// TIA Portal V20 export
// export: Created 2025-12-01T14:56:54.1618983Z, ExportSetting None, DisplayName Totally Integrated Automation Portal, DisplayVersion V20 Update 3, DisplayName TIA Portal Openness, DisplayVersion V20 Update 3, DisplayName TIA Portal Version Control Interface, DisplayVersion V20 Update 3, DisplayName STEP 7 Professional, DisplayVersion V20 Update 3, DisplayName STEP 7 Safety, DisplayVersion V20 Update 2, DisplayName WinCC Basic/Comfort/Advanced, DisplayVersion V20 Update 3, DisplayName WinCC Professional, DisplayVersion V20 Update 3, DisplayName WinCC Unified, DisplayVersion V20 Update 3
FUNCTION_BLOCK "FB341_DesapiladorBandejas_RIANTICS"   // FB341, LAD
{ S7_Optimized_Access := 'FALSE' }
// stored: AutoNumber false, SetENOAutomatically false
   VAR_INPUT
      Maquina : UInt;   // Numero de Maquina (Mesa)
      Error_Tx : Bool;   // Error en el Tx
      EnTension : Bool;   // Existe Tension en la Maquina
      MAQx_Desabilitada : Bool;   // Config MAQ. >>> DesHabilitada
      Termico_Elevacion : Bool;   // Termico de la Elevacion
      PhsMx : Bool;
      Pos_DW : Bool;   // Posición Baja del Apilador
      Pos_MID_DW : Bool;
      Pos_MID_UP : Bool;
      Pos_UP : Bool;   // Posición Alta del Apilador
      EnMovimiento_Elevacion : Bool;   // En Movineto la Elevacion
      CargaSueltaDerecha : Bool;   // Carga Suelta en el Apilador
      CargaSueltaIzquierda : Bool;
      CargaCogidaDerecha : Bool;   // Carga Cogida en el Apilador
      CargaCogidaIzquierda : Bool;
      EnMovimiento_Horquillado : Bool;   // En Movimiento el Hoquillado
      MAQ_DejarBandejas : Bool;   // Interlock >> Dejar Bandejas
      MAQ_CogerBandejas : Bool;   // Interlock >> Coger Bandejas
      MAQ_BuscarCero : Bool;   // Interlock >> Buscar Cero
      CogiendoDerecha : Bool;
      CogiendoIzquierda : Bool;
      DejandoDerecha : Bool;
      DejandoIzquierda : Bool;
      V_TOut_Elevacion : Int := 2000;   // TimeOut del Mov. de Elevacion
      V_TOut_Horquillado : Int := 2000;   // TimeOut del Mov. de Horquillado
   END_VAR
   VAR_OUTPUT
      MAQ_DejadasBandejas : Bool;   // Interlock >> Bandejas Dejadas
      MAQ_CojidasBandejas : Bool;   // Interlock >> Bandejas Cogidas
      MAQ_CeroEncontrado : Bool;   // Interlock >> Bandejas
   END_VAR
   VAR
      AP_ET00 : Bool;
      AP_ET01 : Bool;
      AP_ET100 : Bool;
      AP_ET101 : Bool;
      AP_ET102 : Bool;
      AP_ET103 : Bool;
      AP_ET104 : Bool;
      AP_ET50 : Bool;
      AP_ET51 : Bool;
      AP_ET52 : Bool;
      AP_ET53 : Bool;
      AP_ET60 : Bool;
      AP_ET61 : Bool;
      AP_ET62 : Bool;
      AP_ET63 : Bool;
      AP_ET64 : Bool;
      AP_ET65 : Bool;
      AP_ET66 : Bool;
      MA_Motor_Elev : Bool;
      MA_Slow_Velocity : Bool;
      MA_CogerCarga : Bool;   // Cerrar Cilindros para coger la pila
      MA_DejarCarga : Bool;   // Abrir Cilindros para dejas la pila
      TMP_ReposoCargaSuelta { S7_SetPoint := 'True'} : TON_TIME;
      TMP_EnTension { S7_SetPoint := 'True'} : "FB910_CNT_UHS";
      TOut_Elevacion { S7_SetPoint := 'True'} : "FB910_CNT_UHS";
      TOut_Horquillado { S7_SetPoint := 'True'} : "FB910_CNT_UHS";
      Manual : "MoviManualMaquina_Desapilador_bandejas";
   END_VAR
   VAR_TEMP
      EstadoZona : "EstadoZona";   // Estado de Zona de la Mesa
      EstadoMAQ : "EstadoMaquina_Desapilador_bandejas";   // Estado del Vehiculo Inteliguente de la Maquina
      Aux_ET00 : Bool;
   END_VAR
BEGIN

REGION Network 1: INICIALIZAR - Recoger las Variables de Estado de la Maquina
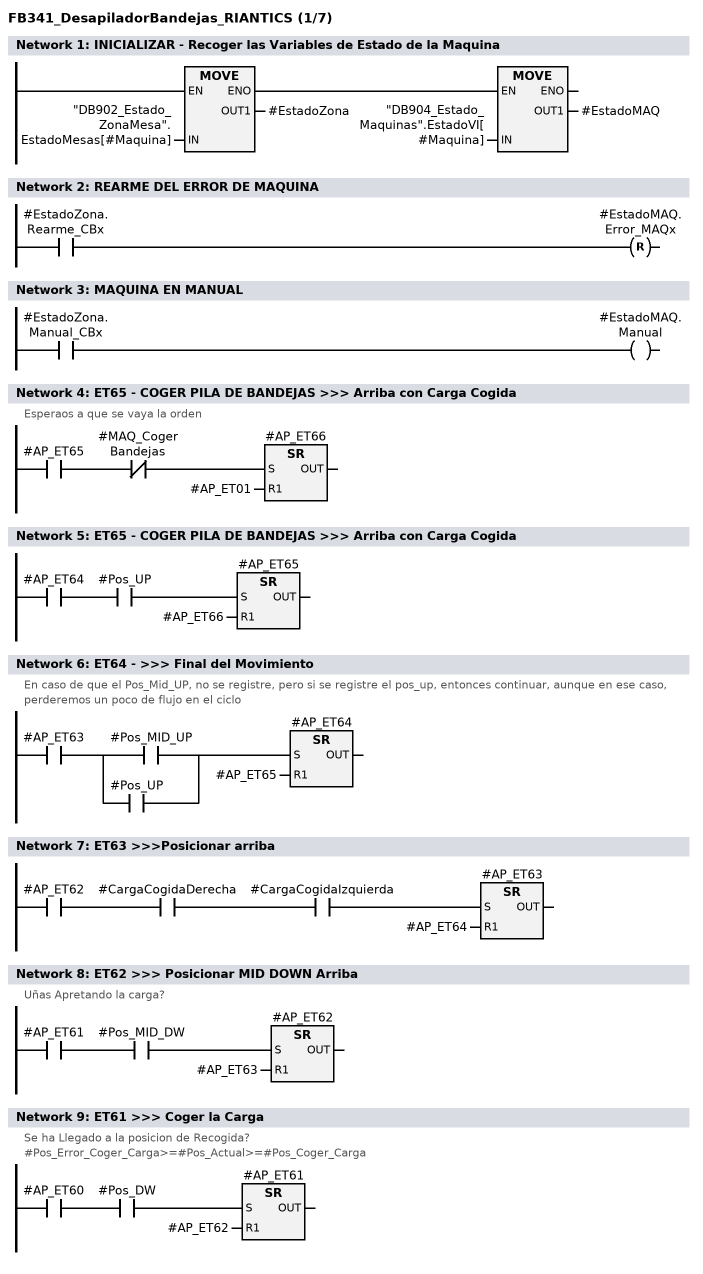
   RUNG wire#powerrail
      Move(in := "DB902_Estado_ZonaMesa".EstadoMesas[#Maquina], out1 => #EstadoZona)
      Move(in := "DB904_Estado_Maquinas".EstadoVI[#Maquina], out1 => #EstadoMAQ)
   END_RUNG
   // the same network as SCL:
   #EstadoZona := "DB902_Estado_ZonaMesa".EstadoMesas[#Maquina];
   #EstadoMAQ := "DB904_Estado_Maquinas".EstadoVI[#Maquina];
END_REGION

REGION Network 2: REARME DEL ERROR DE MAQUINA
   RUNG wire#powerrail
      Contact( #EstadoZona.Rearme_CBx )
      R_Coil( #EstadoMAQ.Error_MAQx )
   END_RUNG
   // the same network as SCL:
   IF #EstadoZona.Rearme_CBx THEN #EstadoMAQ.Error_MAQx := FALSE; END_IF;
END_REGION

REGION Network 3: MAQUINA EN MANUAL
   RUNG wire#powerrail
      Contact( #EstadoZona.Manual_CBx )
      Coil( #EstadoMAQ.Manual )
   END_RUNG
   // the same network as SCL:
   #EstadoMAQ.Manual := #EstadoZona.Manual_CBx;
END_REGION

REGION Network 4: ET65 - COGER PILA DE BANDEJAS >>> Arriba con Carga Cogida
   // Esperaos a que se vaya la orden
   RUNG wire#powerrail
      Contact( #AP_ET65 )
      I_Contact( #MAQ_CogerBandejas )
      S_SR(operand := #AP_ET66, r1 := #AP_ET01)
   END_RUNG
   // the same network as SCL:
   IF #AP_ET65 AND NOT #MAQ_CogerBandejas THEN
       #AP_ET66 := TRUE;   // SR flip-flop
   END_IF;
   IF #AP_ET01 THEN #AP_ET66 := FALSE; END_IF;
END_REGION

REGION Network 5: ET65 - COGER PILA DE BANDEJAS >>> Arriba con Carga Cogida
   RUNG wire#powerrail
      Contact( #AP_ET64 )
      Contact( #Pos_UP )
      S_SR(operand := #AP_ET65, r1 := #AP_ET66)
   END_RUNG
   // the same network as SCL:
   IF #AP_ET64 AND #Pos_UP THEN
       #AP_ET65 := TRUE;   // SR flip-flop
   END_IF;
   IF #AP_ET66 THEN #AP_ET65 := FALSE; END_IF;
END_REGION

REGION Network 6: ET64 - >>> Final del Movimiento
   // En caso de que el Pos_Mid_UP, no se registre, pero si se registre el pos_up, entonces continuar, aunque en ese caso, perderemos un poco de flujo en el ciclo
   RUNG wire#powerrail
      Contact( #AP_ET63 )
      wire#w1
      Contact( #Pos_MID_UP )
      wire#w2
      S_SR(operand := #AP_ET64, r1 := #AP_ET65)
   END_RUNG
   RUNG wire#w1
      Contact( #Pos_UP )
   END_RUNG wire#w2
   // the same network as SCL:
   IF #AP_ET63 AND (#Pos_MID_UP OR #Pos_UP) THEN
       #AP_ET64 := TRUE;   // SR flip-flop
   END_IF;
   IF #AP_ET65 THEN #AP_ET64 := FALSE; END_IF;
END_REGION

REGION Network 7: ET63 >>>Posicionar arriba
   RUNG wire#powerrail
      Contact( #AP_ET62 )
      Contact( #CargaCogidaDerecha )
      Contact( #CargaCogidaIzquierda )
      S_SR(operand := #AP_ET63, r1 := #AP_ET64)
   END_RUNG
   // the same network as SCL:
   IF #AP_ET62 AND #CargaCogidaDerecha AND #CargaCogidaIzquierda THEN
       #AP_ET63 := TRUE;   // SR flip-flop
   END_IF;
   IF #AP_ET64 THEN #AP_ET63 := FALSE; END_IF;
END_REGION

REGION Network 8: ET62 >>> Posicionar MID DOWN Arriba
   // Uñas Apretando la carga?
   RUNG wire#powerrail
      Contact( #AP_ET61 )
      Contact( #Pos_MID_DW )
      S_SR(operand := #AP_ET62, r1 := #AP_ET63)
   END_RUNG
   // the same network as SCL:
   IF #AP_ET61 AND #Pos_MID_DW THEN
       #AP_ET62 := TRUE;   // SR flip-flop
   END_IF;
   IF #AP_ET63 THEN #AP_ET62 := FALSE; END_IF;
END_REGION

REGION Network 9: ET61 >>> Coger la Carga
   // Se ha Llegado a la posicion de Recogida?
   // #Pos_Error_Coger_Carga>=#Pos_Actual>=#Pos_Coger_Carga
   RUNG wire#powerrail
      Contact( #AP_ET60 )
      Contact( #Pos_DW )
      S_SR(operand := #AP_ET61, r1 := #AP_ET62)
   END_RUNG
   // the same network as SCL:
   IF #AP_ET60 AND #Pos_DW THEN
       #AP_ET61 := TRUE;   // SR flip-flop
   END_IF;
   IF #AP_ET62 THEN #AP_ET61 := FALSE; END_IF;
END_REGION

REGION Network 10: ET60 >>> Posicionar Abajo(Anulado)
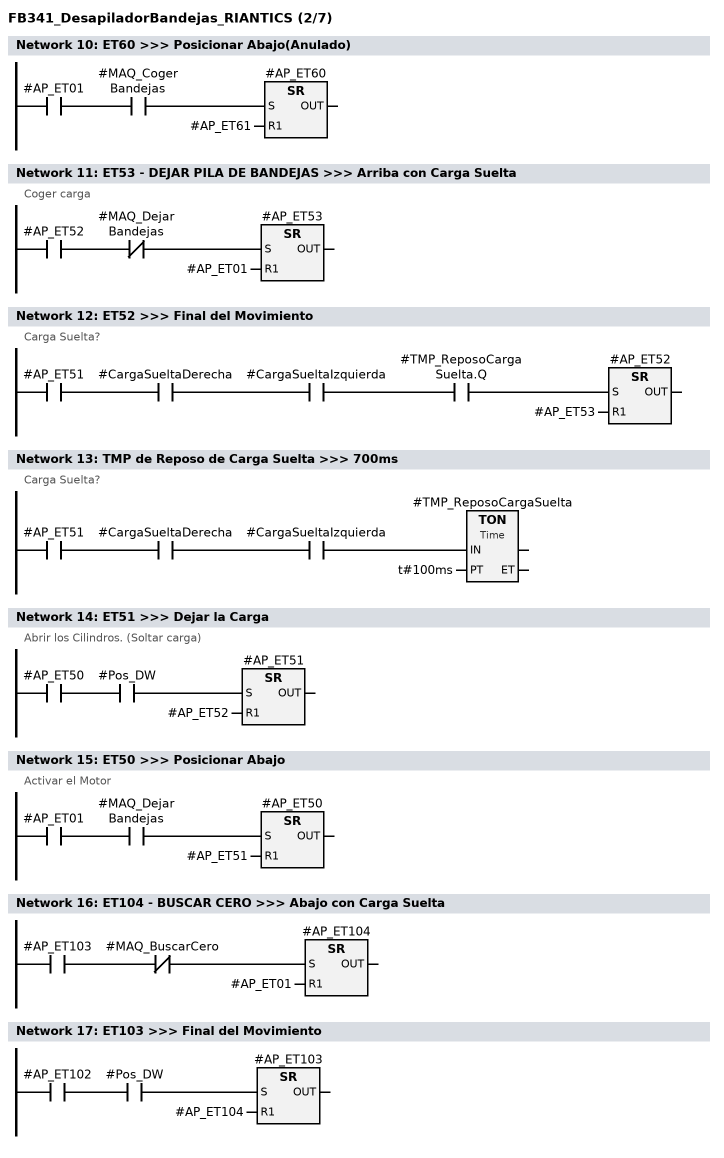
   RUNG wire#powerrail
      Contact( #AP_ET01 )
      Contact( #MAQ_CogerBandejas )
      S_SR(operand := #AP_ET60, r1 := #AP_ET61)
   END_RUNG
   // the same network as SCL:
   IF #AP_ET01 AND #MAQ_CogerBandejas THEN
       #AP_ET60 := TRUE;   // SR flip-flop
   END_IF;
   IF #AP_ET61 THEN #AP_ET60 := FALSE; END_IF;
END_REGION

REGION Network 11: ET53 - DEJAR PILA DE BANDEJAS >>> Arriba con Carga Suelta
   // Coger carga
   RUNG wire#powerrail
      Contact( #AP_ET52 )
      I_Contact( #MAQ_DejarBandejas )
      S_SR(operand := #AP_ET53, r1 := #AP_ET01)
   END_RUNG
   // the same network as SCL:
   IF #AP_ET52 AND NOT #MAQ_DejarBandejas THEN
       #AP_ET53 := TRUE;   // SR flip-flop
   END_IF;
   IF #AP_ET01 THEN #AP_ET53 := FALSE; END_IF;
END_REGION

REGION Network 12: ET52 >>> Final del Movimiento
   // Carga Suelta?
   RUNG wire#powerrail
      Contact( #AP_ET51 )
      Contact( #CargaSueltaDerecha )
      Contact( #CargaSueltaIzquierda )
      Contact( #TMP_ReposoCargaSuelta.Q )
      S_SR(operand := #AP_ET52, r1 := #AP_ET53)
   END_RUNG
   // the same network as SCL:
   IF #AP_ET51 AND #CargaSueltaDerecha AND #CargaSueltaIzquierda AND #TMP_ReposoCargaSuelta.Q THEN
       #AP_ET52 := TRUE;   // SR flip-flop
   END_IF;
   IF #AP_ET53 THEN #AP_ET52 := FALSE; END_IF;
END_REGION

REGION Network 13: TMP de Reposo de Carga Suelta >>> 700ms
   // Carga Suelta?
   RUNG wire#powerrail
      Contact( #AP_ET51 )
      Contact( #CargaSueltaDerecha )
      Contact( #CargaSueltaIzquierda )
      { S7_Templates := "time_type := Time" } #TMP_ReposoCargaSuelta.TON(pt := t#100ms, et =>)
   END_RUNG
   // the same network as SCL:
   #TMP_ReposoCargaSuelta(IN := #AP_ET51 AND #CargaSueltaDerecha AND #CargaSueltaIzquierda, PT := t#100ms);   // TON
END_REGION

REGION Network 14: ET51 >>> Dejar la Carga
   // Abrir los Cilindros. (Soltar carga)
   RUNG wire#powerrail
      Contact( #AP_ET50 )
      Contact( #Pos_DW )
      S_SR(operand := #AP_ET51, r1 := #AP_ET52)
   END_RUNG
   // the same network as SCL:
   IF #AP_ET50 AND #Pos_DW THEN
       #AP_ET51 := TRUE;   // SR flip-flop
   END_IF;
   IF #AP_ET52 THEN #AP_ET51 := FALSE; END_IF;
END_REGION

REGION Network 15: ET50 >>> Posicionar Abajo
   // Activar el Motor
   RUNG wire#powerrail
      Contact( #AP_ET01 )
      Contact( #MAQ_DejarBandejas )
      S_SR(operand := #AP_ET50, r1 := #AP_ET51)
   END_RUNG
   // the same network as SCL:
   IF #AP_ET01 AND #MAQ_DejarBandejas THEN
       #AP_ET50 := TRUE;   // SR flip-flop
   END_IF;
   IF #AP_ET51 THEN #AP_ET50 := FALSE; END_IF;
END_REGION

REGION Network 16: ET104 - BUSCAR CERO >>> Abajo con Carga Suelta
   RUNG wire#powerrail
      Contact( #AP_ET103 )
      I_Contact( #MAQ_BuscarCero )
      S_SR(operand := #AP_ET104, r1 := #AP_ET01)
   END_RUNG
   // the same network as SCL:
   IF #AP_ET103 AND NOT #MAQ_BuscarCero THEN
       #AP_ET104 := TRUE;   // SR flip-flop
   END_IF;
   IF #AP_ET01 THEN #AP_ET104 := FALSE; END_IF;
END_REGION

REGION Network 17: ET103 >>> Final del Movimiento
   RUNG wire#powerrail
      Contact( #AP_ET102 )
      Contact( #Pos_DW )
      S_SR(operand := #AP_ET103, r1 := #AP_ET104)
   END_RUNG
   // the same network as SCL:
   IF #AP_ET102 AND #Pos_DW THEN
       #AP_ET103 := TRUE;   // SR flip-flop
   END_IF;
   IF #AP_ET104 THEN #AP_ET103 := FALSE; END_IF;
END_REGION

REGION Network 18: ET102 >>> Posicionar Abajo
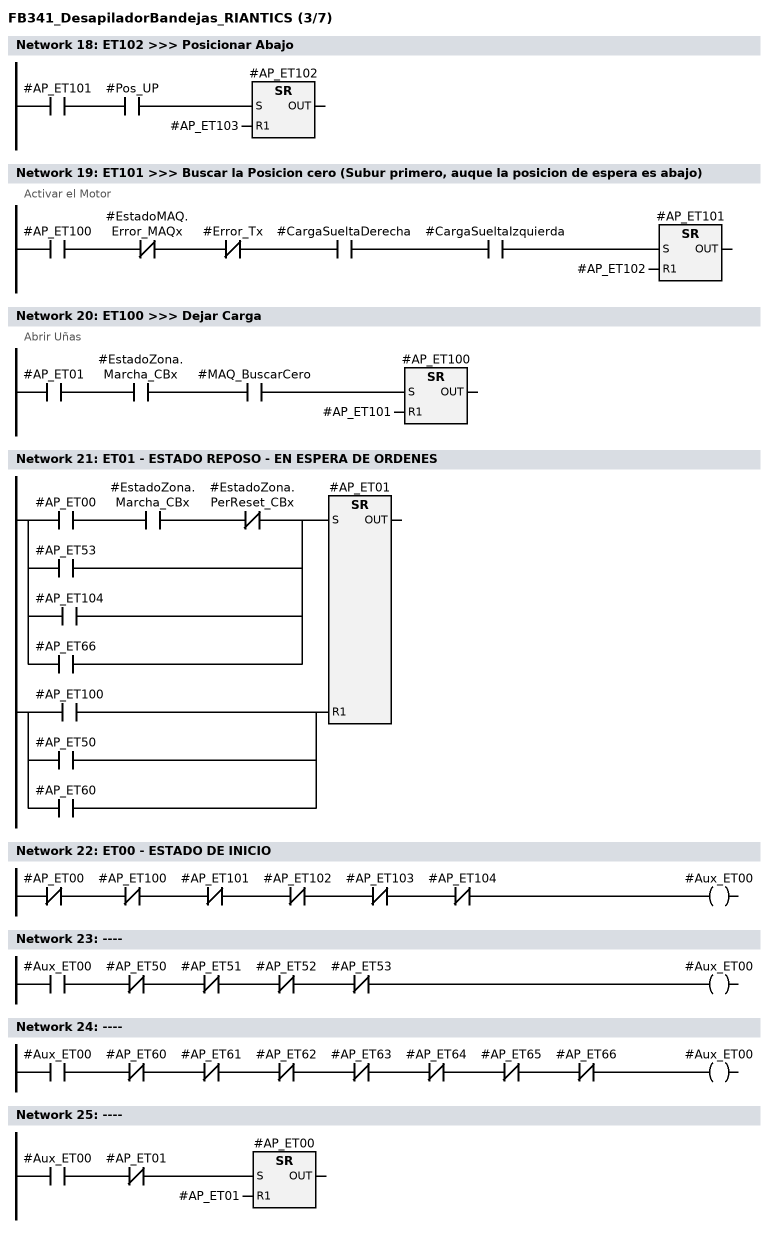
   RUNG wire#powerrail
      Contact( #AP_ET101 )
      Contact( #Pos_UP )
      S_SR(operand := #AP_ET102, r1 := #AP_ET103)
   END_RUNG
   // the same network as SCL:
   IF #AP_ET101 AND #Pos_UP THEN
       #AP_ET102 := TRUE;   // SR flip-flop
   END_IF;
   IF #AP_ET103 THEN #AP_ET102 := FALSE; END_IF;
END_REGION

REGION Network 19: ET101 >>> Buscar la Posicion cero (Subur primero, auque la posicion de espera es abajo)
   // Activar el Motor
   RUNG wire#powerrail
      Contact( #AP_ET100 )
      I_Contact( #EstadoMAQ.Error_MAQx )
      I_Contact( #Error_Tx )
      Contact( #CargaSueltaDerecha )
      Contact( #CargaSueltaIzquierda )
      S_SR(operand := #AP_ET101, r1 := #AP_ET102)
   END_RUNG
   // the same network as SCL:
   IF #AP_ET100 AND NOT #EstadoMAQ.Error_MAQx AND NOT #Error_Tx AND #CargaSueltaDerecha AND #CargaSueltaIzquierda THEN
       #AP_ET101 := TRUE;   // SR flip-flop
   END_IF;
   IF #AP_ET102 THEN #AP_ET101 := FALSE; END_IF;
END_REGION

REGION Network 20: ET100 >>> Dejar Carga
   // Abrir Uñas
   RUNG wire#powerrail
      Contact( #AP_ET01 )
      Contact( #EstadoZona.Marcha_CBx )
      Contact( #MAQ_BuscarCero )
      S_SR(operand := #AP_ET100, r1 := #AP_ET101)
   END_RUNG
   // the same network as SCL:
   IF #AP_ET01 AND #EstadoZona.Marcha_CBx AND #MAQ_BuscarCero THEN
       #AP_ET100 := TRUE;   // SR flip-flop
   END_IF;
   IF #AP_ET101 THEN #AP_ET100 := FALSE; END_IF;
END_REGION

REGION Network 21: ET01 - ESTADO REPOSO - EN ESPERA DE ORDENES
   RUNG wire#powerrail
      Contact( #AP_ET00 )
      Contact( #EstadoZona.Marcha_CBx )
      I_Contact( #EstadoZona.PerReset_CBx )
      wire#w1
      S_SR(operand := #AP_ET01, r1 := wire#w2)
   END_RUNG
   RUNG wire#powerrail
      Contact( #AP_ET53 )
   END_RUNG wire#w1
   RUNG wire#powerrail
      Contact( #AP_ET104 )
   END_RUNG wire#w1
   RUNG wire#powerrail
      Contact( #AP_ET66 )
   END_RUNG wire#w1
   RUNG wire#powerrail
      Contact( #AP_ET100 )
   END_RUNG wire#w2
   RUNG wire#powerrail
      Contact( #AP_ET50 )
   END_RUNG wire#w2
   RUNG wire#powerrail
      Contact( #AP_ET60 )
   END_RUNG wire#w2
   // the same network as SCL:
   IF (#AP_ET00 AND #EstadoZona.Marcha_CBx AND NOT #EstadoZona.PerReset_CBx) OR #AP_ET53 OR #AP_ET104 OR #AP_ET66 THEN
       #AP_ET01 := TRUE;   // SR flip-flop
   END_IF;
   IF #AP_ET100 OR #AP_ET50 OR #AP_ET60 THEN #AP_ET01 := FALSE; END_IF;
END_REGION

REGION Network 22: ET00 - ESTADO DE INICIO
   RUNG wire#powerrail
      I_Contact( #AP_ET00 )
      I_Contact( #AP_ET100 )
      I_Contact( #AP_ET101 )
      I_Contact( #AP_ET102 )
      I_Contact( #AP_ET103 )
      I_Contact( #AP_ET104 )
      Coil( #Aux_ET00 )
   END_RUNG
   // the same network as SCL:
   #Aux_ET00 := NOT #AP_ET00 AND NOT #AP_ET100 AND NOT #AP_ET101 AND NOT #AP_ET102 AND NOT #AP_ET103 AND NOT #AP_ET104;
END_REGION

REGION Network 23: ----
   RUNG wire#powerrail
      Contact( #Aux_ET00 )
      I_Contact( #AP_ET50 )
      I_Contact( #AP_ET51 )
      I_Contact( #AP_ET52 )
      I_Contact( #AP_ET53 )
      Coil( #Aux_ET00 )
   END_RUNG
   // the same network as SCL:
   #Aux_ET00 := #Aux_ET00 AND NOT #AP_ET50 AND NOT #AP_ET51 AND NOT #AP_ET52 AND NOT #AP_ET53;
END_REGION

REGION Network 24: ----
   RUNG wire#powerrail
      Contact( #Aux_ET00 )
      I_Contact( #AP_ET60 )
      I_Contact( #AP_ET61 )
      I_Contact( #AP_ET62 )
      I_Contact( #AP_ET63 )
      I_Contact( #AP_ET64 )
      I_Contact( #AP_ET65 )
      I_Contact( #AP_ET66 )
      Coil( #Aux_ET00 )
   END_RUNG
   // the same network as SCL:
   #Aux_ET00 := #Aux_ET00 AND NOT #AP_ET60 AND NOT #AP_ET61 AND NOT #AP_ET62 AND NOT #AP_ET63 AND NOT #AP_ET64 AND NOT #AP_ET65 AND NOT #AP_ET66;
END_REGION

REGION Network 25: ----
   RUNG wire#powerrail
      Contact( #Aux_ET00 )
      I_Contact( #AP_ET01 )
      S_SR(operand := #AP_ET00, r1 := #AP_ET01)
   END_RUNG
   // the same network as SCL:
   IF #Aux_ET00 AND NOT #AP_ET01 THEN
       #AP_ET00 := TRUE;   // SR flip-flop
   END_IF;
   IF #AP_ET01 THEN #AP_ET00 := FALSE; END_IF;
END_REGION

REGION Network 26: INTERLOCK - Dejada la Pila de Bandejas Sobre Bandeja
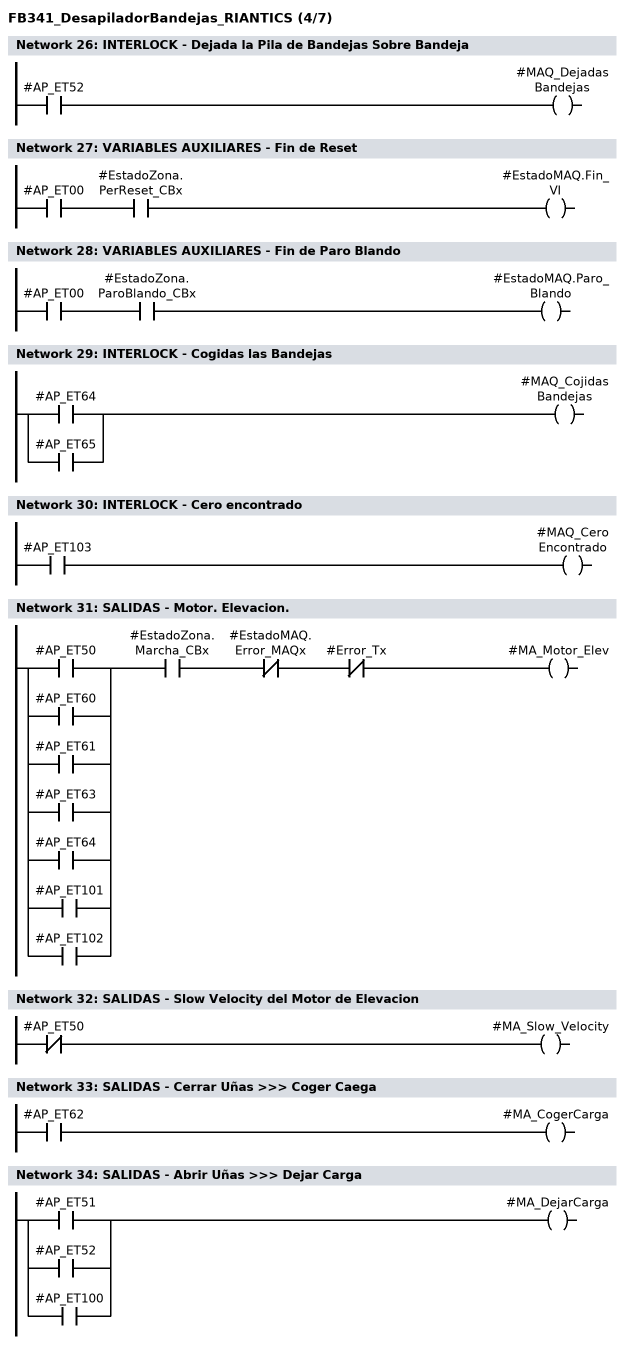
   RUNG wire#powerrail
      Contact( #AP_ET52 )
      Coil( #MAQ_DejadasBandejas )
   END_RUNG
   // the same network as SCL:
   #MAQ_DejadasBandejas := #AP_ET52;
END_REGION

REGION Network 27: VARIABLES AUXILIARES - Fin de Reset
   RUNG wire#powerrail
      Contact( #AP_ET00 )
      Contact( #EstadoZona.PerReset_CBx )
      Coil( #EstadoMAQ.Fin_VI )
   END_RUNG
   // the same network as SCL:
   #EstadoMAQ.Fin_VI := #AP_ET00 AND #EstadoZona.PerReset_CBx;
END_REGION

REGION Network 28: VARIABLES AUXILIARES - Fin de Paro Blando
   RUNG wire#powerrail
      Contact( #AP_ET00 )
      Contact( #EstadoZona.ParoBlando_CBx )
      Coil( #EstadoMAQ.Paro_Blando )
   END_RUNG
   // the same network as SCL:
   #EstadoMAQ.Paro_Blando := #AP_ET00 AND #EstadoZona.ParoBlando_CBx;
END_REGION

REGION Network 29: INTERLOCK - Cogidas las Bandejas
   RUNG wire#powerrail
      Contact( #AP_ET64 )
      wire#w1
      Coil( #MAQ_CojidasBandejas )
   END_RUNG
   RUNG wire#powerrail
      Contact( #AP_ET65 )
   END_RUNG wire#w1
   // the same network as SCL:
   #MAQ_CojidasBandejas := #AP_ET64 OR #AP_ET65;
END_REGION

REGION Network 30: INTERLOCK - Cero encontrado
   RUNG wire#powerrail
      Contact( #AP_ET103 )
      Coil( #MAQ_CeroEncontrado )
   END_RUNG
   // the same network as SCL:
   #MAQ_CeroEncontrado := #AP_ET103;
END_REGION

REGION Network 31: SALIDAS - Motor. Elevacion.
   RUNG wire#powerrail
      Contact( #AP_ET50 )
      wire#w1
      Contact( #EstadoZona.Marcha_CBx )
      I_Contact( #EstadoMAQ.Error_MAQx )
      I_Contact( #Error_Tx )
      Coil( #MA_Motor_Elev )
   END_RUNG
   RUNG wire#powerrail
      Contact( #AP_ET60 )
   END_RUNG wire#w1
   RUNG wire#powerrail
      Contact( #AP_ET61 )
   END_RUNG wire#w1
   RUNG wire#powerrail
      Contact( #AP_ET63 )
   END_RUNG wire#w1
   RUNG wire#powerrail
      Contact( #AP_ET64 )
   END_RUNG wire#w1
   RUNG wire#powerrail
      Contact( #AP_ET101 )
   END_RUNG wire#w1
   RUNG wire#powerrail
      Contact( #AP_ET102 )
   END_RUNG wire#w1
   // the same network as SCL:
   #MA_Motor_Elev := (#AP_ET50 OR #AP_ET60 OR #AP_ET61 OR #AP_ET63 OR #AP_ET64 OR #AP_ET101 OR #AP_ET102) AND #EstadoZona.Marcha_CBx AND NOT #EstadoMAQ.Error_MAQx AND NOT #Error_Tx;
END_REGION

REGION Network 32: SALIDAS - Slow Velocity del Motor de Elevacion
   RUNG wire#powerrail
      I_Contact( #AP_ET50 )
      Coil( #MA_Slow_Velocity )
   END_RUNG
   // the same network as SCL:
   #MA_Slow_Velocity := NOT #AP_ET50;
END_REGION

REGION Network 33: SALIDAS - Cerrar Uñas >>> Coger Caega
   RUNG wire#powerrail
      Contact( #AP_ET62 )
      Coil( #MA_CogerCarga )
   END_RUNG
   // the same network as SCL:
   #MA_CogerCarga := #AP_ET62;
END_REGION

REGION Network 34: SALIDAS - Abrir Uñas >>> Dejar Carga
   RUNG wire#powerrail
      Contact( #AP_ET51 )
      wire#w1
      Coil( #MA_DejarCarga )
   END_RUNG
   RUNG wire#powerrail
      Contact( #AP_ET52 )
   END_RUNG wire#w1
   RUNG wire#powerrail
      Contact( #AP_ET100 )
   END_RUNG wire#w1
   // the same network as SCL:
   #MA_DejarCarga := #AP_ET51 OR #AP_ET52 OR #AP_ET100;
END_REGION

REGION Network 35: TMP - Espera En Tension
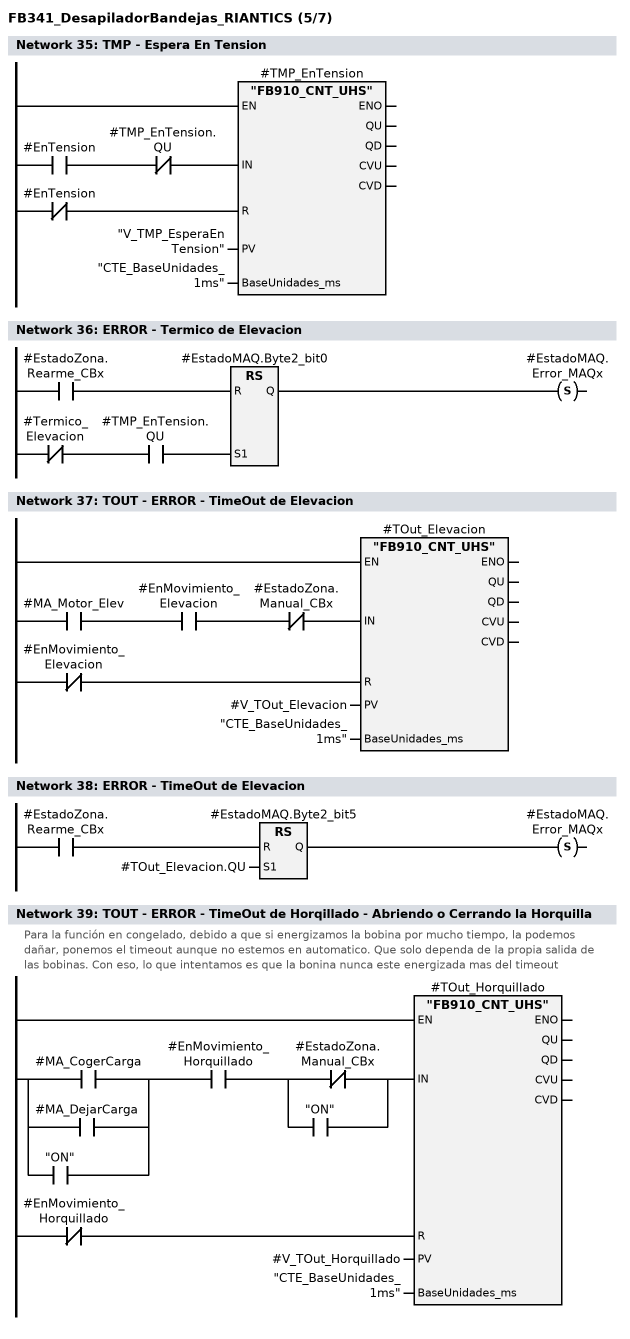
   RUNG wire#powerrail
      #TMP_EnTension(IN := wire#w1, R := wire#w2, PV := "V_TMP_EsperaEnTension", BaseUnidades_ms := "CTE_BaseUnidades_1ms", QU =>, QD =>, CVU =>, CVD =>)
   END_RUNG
   RUNG wire#powerrail
      Contact( #EnTension )
      I_Contact( #TMP_EnTension.QU )
   END_RUNG wire#w1
   RUNG wire#powerrail
      I_Contact( #EnTension )
   END_RUNG wire#w2
   // the same network as SCL:
   #TMP_EnTension(IN := #EnTension AND NOT #TMP_EnTension.QU,   // "FB910_CNT_UHS"
                  R := NOT #EnTension,
                  PV := "V_TMP_EsperaEnTension",
                  BaseUnidades_ms := "CTE_BaseUnidades_1ms");
END_REGION

REGION Network 36: ERROR - Termico de Elevacion
   RUNG wire#powerrail
      Contact( #EstadoZona.Rearme_CBx )
      S_RS(operand := #EstadoMAQ.Byte2_bit0, s1 := wire#w1)
      S_Coil( #EstadoMAQ.Error_MAQx )
   END_RUNG
   RUNG wire#powerrail
      I_Contact( #Termico_Elevacion )
      Contact( #TMP_EnTension.QU )
   END_RUNG wire#w1
   // the same network as SCL:
   IF #EstadoZona.Rearme_CBx THEN
       #EstadoMAQ.Byte2_bit0 := FALSE;   // RS flip-flop
   END_IF;
   IF NOT #Termico_Elevacion AND #TMP_EnTension.QU THEN #EstadoMAQ.Byte2_bit0 := TRUE; END_IF;
   IF #EstadoMAQ.Byte2_bit0 THEN #EstadoMAQ.Error_MAQx := TRUE; END_IF;
END_REGION

REGION Network 37: TOUT - ERROR - TimeOut de Elevacion
   RUNG wire#powerrail
      #TOut_Elevacion(IN := wire#w1, R := wire#w2, PV := #V_TOut_Elevacion, BaseUnidades_ms := "CTE_BaseUnidades_1ms", QU =>, QD =>, CVU =>, CVD =>)
   END_RUNG
   RUNG wire#powerrail
      Contact( #MA_Motor_Elev )
      Contact( #EnMovimiento_Elevacion )
      I_Contact( #EstadoZona.Manual_CBx )
   END_RUNG wire#w1
   RUNG wire#powerrail
      I_Contact( #EnMovimiento_Elevacion )
   END_RUNG wire#w2
   // the same network as SCL:
   #TOut_Elevacion(IN := #MA_Motor_Elev AND #EnMovimiento_Elevacion AND NOT #EstadoZona.Manual_CBx,   // "FB910_CNT_UHS"
                   R := NOT #EnMovimiento_Elevacion,
                   PV := #V_TOut_Elevacion,
                   BaseUnidades_ms := "CTE_BaseUnidades_1ms");
END_REGION

REGION Network 38: ERROR - TimeOut de Elevacion
   RUNG wire#powerrail
      Contact( #EstadoZona.Rearme_CBx )
      S_RS(operand := #EstadoMAQ.Byte2_bit5, s1 := #TOut_Elevacion.QU)
      S_Coil( #EstadoMAQ.Error_MAQx )
   END_RUNG
   // the same network as SCL:
   IF #EstadoZona.Rearme_CBx THEN
       #EstadoMAQ.Byte2_bit5 := FALSE;   // RS flip-flop
   END_IF;
   IF #TOut_Elevacion.QU THEN #EstadoMAQ.Byte2_bit5 := TRUE; END_IF;
   IF #EstadoMAQ.Byte2_bit5 THEN #EstadoMAQ.Error_MAQx := TRUE; END_IF;
END_REGION

REGION Network 39: TOUT - ERROR - TimeOut de Horqillado - Abriendo o Cerrando la Horquilla
   // Para la función en congelado, debido a que si energizamos la bobina por mucho tiempo, la podemos dañar, ponemos el timeout aunque no estemos en automatico. Que solo dependa de la propia salida de las bobinas. Con eso, lo que intentamos es que la bonina nunca este energizada mas del timeout
   RUNG wire#powerrail
      #TOut_Horquillado(IN := wire#w3, R := wire#w4, PV := #V_TOut_Horquillado, BaseUnidades_ms := "CTE_BaseUnidades_1ms", QU =>, QD =>, CVU =>, CVD =>)
   END_RUNG
   RUNG wire#powerrail
      Contact( #MA_CogerCarga )
      wire#w1
      Contact( #EnMovimiento_Horquillado )
      wire#w2
      I_Contact( #EstadoZona.Manual_CBx )
   END_RUNG wire#w3
   RUNG wire#powerrail
      Contact( #MA_DejarCarga )
   END_RUNG wire#w1
   RUNG wire#powerrail
      Contact( "ON" )
   END_RUNG wire#w1
   RUNG wire#w2
      Contact( "ON" )
   END_RUNG wire#w3
   RUNG wire#powerrail
      I_Contact( #EnMovimiento_Horquillado )
   END_RUNG wire#w4
   // the same network as SCL:
   #TOut_Horquillado(IN := (#MA_CogerCarga OR #MA_DejarCarga OR "ON") AND #EnMovimiento_Horquillado AND (NOT #EstadoZona.Manual_CBx OR "ON"),   // "FB910_CNT_UHS"
                     R := NOT #EnMovimiento_Horquillado,
                     PV := #V_TOut_Horquillado,
                     BaseUnidades_ms := "CTE_BaseUnidades_1ms");
END_REGION

REGION Network 40: ERROR - TimeOut de Horqillado - Abriendo la Horquilla Izquierda
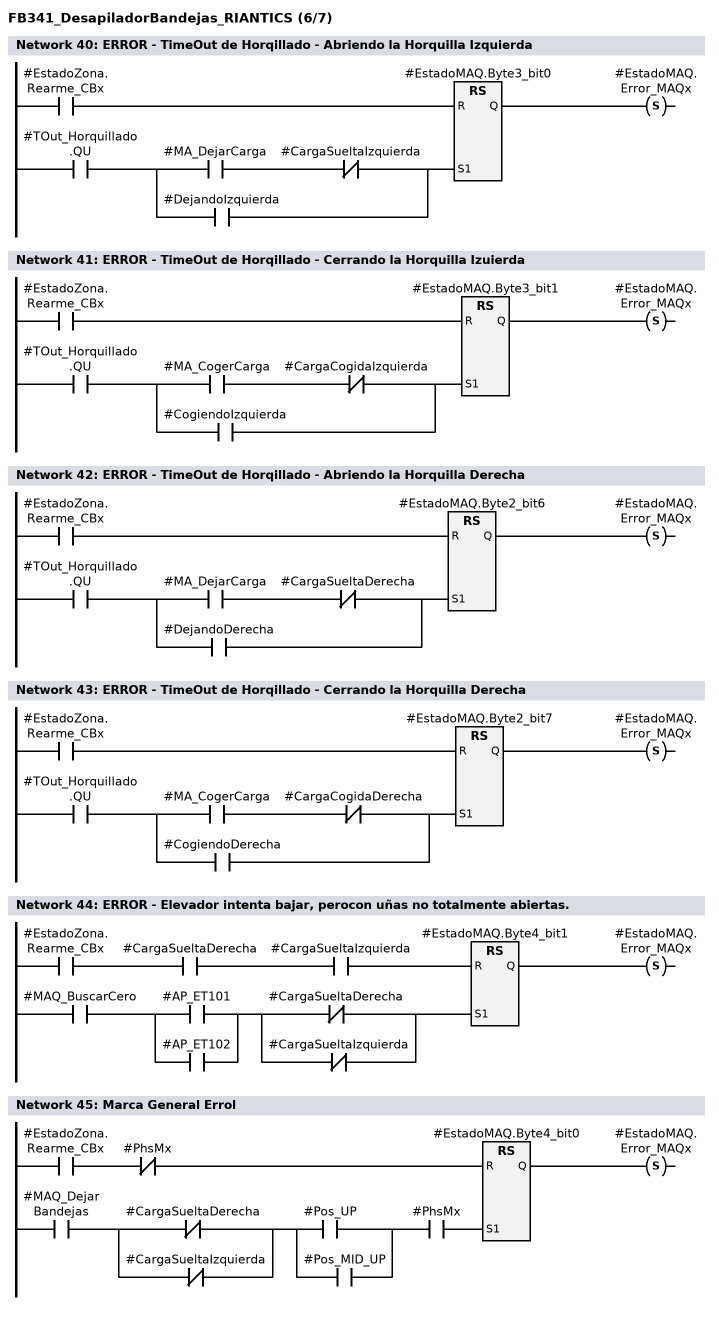
   RUNG wire#powerrail
      Contact( #EstadoZona.Rearme_CBx )
      S_RS(operand := #EstadoMAQ.Byte3_bit0, s1 := wire#w2)
      S_Coil( #EstadoMAQ.Error_MAQx )
   END_RUNG
   RUNG wire#powerrail
      Contact( #TOut_Horquillado.QU )
      wire#w1
      Contact( #MA_DejarCarga )
      I_Contact( #CargaSueltaIzquierda )
   END_RUNG wire#w2
   RUNG wire#w1
      Contact( #DejandoIzquierda )
   END_RUNG wire#w2
   // the same network as SCL:
   IF #EstadoZona.Rearme_CBx THEN
       #EstadoMAQ.Byte3_bit0 := FALSE;   // RS flip-flop
   END_IF;
   IF #TOut_Horquillado.QU AND ((#MA_DejarCarga AND NOT #CargaSueltaIzquierda) OR #DejandoIzquierda) THEN
       #EstadoMAQ.Byte3_bit0 := TRUE;
   END_IF;
   IF #EstadoMAQ.Byte3_bit0 THEN #EstadoMAQ.Error_MAQx := TRUE; END_IF;
END_REGION

REGION Network 41: ERROR - TimeOut de Horqillado - Cerrando la Horquilla Izuierda
   RUNG wire#powerrail
      Contact( #EstadoZona.Rearme_CBx )
      S_RS(operand := #EstadoMAQ.Byte3_bit1, s1 := wire#w2)
      S_Coil( #EstadoMAQ.Error_MAQx )
   END_RUNG
   RUNG wire#powerrail
      Contact( #TOut_Horquillado.QU )
      wire#w1
      Contact( #MA_CogerCarga )
      I_Contact( #CargaCogidaIzquierda )
   END_RUNG wire#w2
   RUNG wire#w1
      Contact( #CogiendoIzquierda )
   END_RUNG wire#w2
   // the same network as SCL:
   IF #EstadoZona.Rearme_CBx THEN
       #EstadoMAQ.Byte3_bit1 := FALSE;   // RS flip-flop
   END_IF;
   IF #TOut_Horquillado.QU AND ((#MA_CogerCarga AND NOT #CargaCogidaIzquierda) OR #CogiendoIzquierda) THEN
       #EstadoMAQ.Byte3_bit1 := TRUE;
   END_IF;
   IF #EstadoMAQ.Byte3_bit1 THEN #EstadoMAQ.Error_MAQx := TRUE; END_IF;
END_REGION

REGION Network 42: ERROR - TimeOut de Horqillado - Abriendo la Horquilla Derecha
   RUNG wire#powerrail
      Contact( #EstadoZona.Rearme_CBx )
      S_RS(operand := #EstadoMAQ.Byte2_bit6, s1 := wire#w2)
      S_Coil( #EstadoMAQ.Error_MAQx )
   END_RUNG
   RUNG wire#powerrail
      Contact( #TOut_Horquillado.QU )
      wire#w1
      Contact( #MA_DejarCarga )
      I_Contact( #CargaSueltaDerecha )
   END_RUNG wire#w2
   RUNG wire#w1
      Contact( #DejandoDerecha )
   END_RUNG wire#w2
   // the same network as SCL:
   IF #EstadoZona.Rearme_CBx THEN
       #EstadoMAQ.Byte2_bit6 := FALSE;   // RS flip-flop
   END_IF;
   IF #TOut_Horquillado.QU AND ((#MA_DejarCarga AND NOT #CargaSueltaDerecha) OR #DejandoDerecha) THEN
       #EstadoMAQ.Byte2_bit6 := TRUE;
   END_IF;
   IF #EstadoMAQ.Byte2_bit6 THEN #EstadoMAQ.Error_MAQx := TRUE; END_IF;
END_REGION

REGION Network 43: ERROR - TimeOut de Horqillado - Cerrando la Horquilla Derecha
   RUNG wire#powerrail
      Contact( #EstadoZona.Rearme_CBx )
      S_RS(operand := #EstadoMAQ.Byte2_bit7, s1 := wire#w2)
      S_Coil( #EstadoMAQ.Error_MAQx )
   END_RUNG
   RUNG wire#powerrail
      Contact( #TOut_Horquillado.QU )
      wire#w1
      Contact( #MA_CogerCarga )
      I_Contact( #CargaCogidaDerecha )
   END_RUNG wire#w2
   RUNG wire#w1
      Contact( #CogiendoDerecha )
   END_RUNG wire#w2
   // the same network as SCL:
   IF #EstadoZona.Rearme_CBx THEN
       #EstadoMAQ.Byte2_bit7 := FALSE;   // RS flip-flop
   END_IF;
   IF #TOut_Horquillado.QU AND ((#MA_CogerCarga AND NOT #CargaCogidaDerecha) OR #CogiendoDerecha) THEN
       #EstadoMAQ.Byte2_bit7 := TRUE;
   END_IF;
   IF #EstadoMAQ.Byte2_bit7 THEN #EstadoMAQ.Error_MAQx := TRUE; END_IF;
END_REGION

REGION Network 44: ERROR - Elevador intenta bajar, perocon uñas no totalmente abiertas.
   RUNG wire#powerrail
      Contact( #EstadoZona.Rearme_CBx )
      Contact( #CargaSueltaDerecha )
      Contact( #CargaSueltaIzquierda )
      S_RS(operand := #EstadoMAQ.Byte4_bit1, s1 := wire#w3)
      S_Coil( #EstadoMAQ.Error_MAQx )
   END_RUNG
   RUNG wire#powerrail
      Contact( #MAQ_BuscarCero )
      wire#w1
      Contact( #AP_ET101 )
      wire#w2
      I_Contact( #CargaSueltaDerecha )
   END_RUNG wire#w3
   RUNG wire#w1
      Contact( #AP_ET102 )
   END_RUNG wire#w2
   RUNG wire#w2
      I_Contact( #CargaSueltaIzquierda )
   END_RUNG wire#w3
   // the same network as SCL:
   IF #EstadoZona.Rearme_CBx AND #CargaSueltaDerecha AND #CargaSueltaIzquierda THEN
       #EstadoMAQ.Byte4_bit1 := FALSE;   // RS flip-flop
   END_IF;
   IF #MAQ_BuscarCero AND (#AP_ET101 OR #AP_ET102) AND (NOT #CargaSueltaDerecha OR NOT #CargaSueltaIzquierda) THEN
       #EstadoMAQ.Byte4_bit1 := TRUE;
   END_IF;
   IF #EstadoMAQ.Byte4_bit1 THEN #EstadoMAQ.Error_MAQx := TRUE; END_IF;
END_REGION

REGION Network 45: Marca General Errol
   RUNG wire#powerrail
      Contact( #EstadoZona.Rearme_CBx )
      I_Contact( #PhsMx )
      S_RS(operand := #EstadoMAQ.Byte4_bit0, s1 := wire#w4)
      S_Coil( #EstadoMAQ.Error_MAQx )
   END_RUNG
   RUNG wire#powerrail
      Contact( #MAQ_DejarBandejas )
      wire#w1
      I_Contact( #CargaSueltaDerecha )
      wire#w2
      Contact( #Pos_UP )
      wire#w3
      Contact( #PhsMx )
   END_RUNG wire#w4
   RUNG wire#w1
      I_Contact( #CargaSueltaIzquierda )
   END_RUNG wire#w2
   RUNG wire#w2
      Contact( #Pos_MID_UP )
   END_RUNG wire#w3
   // the same network as SCL:
   IF #EstadoZona.Rearme_CBx AND NOT #PhsMx THEN
       #EstadoMAQ.Byte4_bit0 := FALSE;   // RS flip-flop
   END_IF;
   IF #MAQ_DejarBandejas AND (NOT #CargaSueltaDerecha OR NOT #CargaSueltaIzquierda) AND (#Pos_UP OR #Pos_MID_UP) AND #PhsMx THEN
       #EstadoMAQ.Byte4_bit0 := TRUE;
   END_IF;
   IF #EstadoMAQ.Byte4_bit0 THEN #EstadoMAQ.Error_MAQx := TRUE; END_IF;
END_REGION

REGION Network 46: ESTADO DE LA MAQUINA
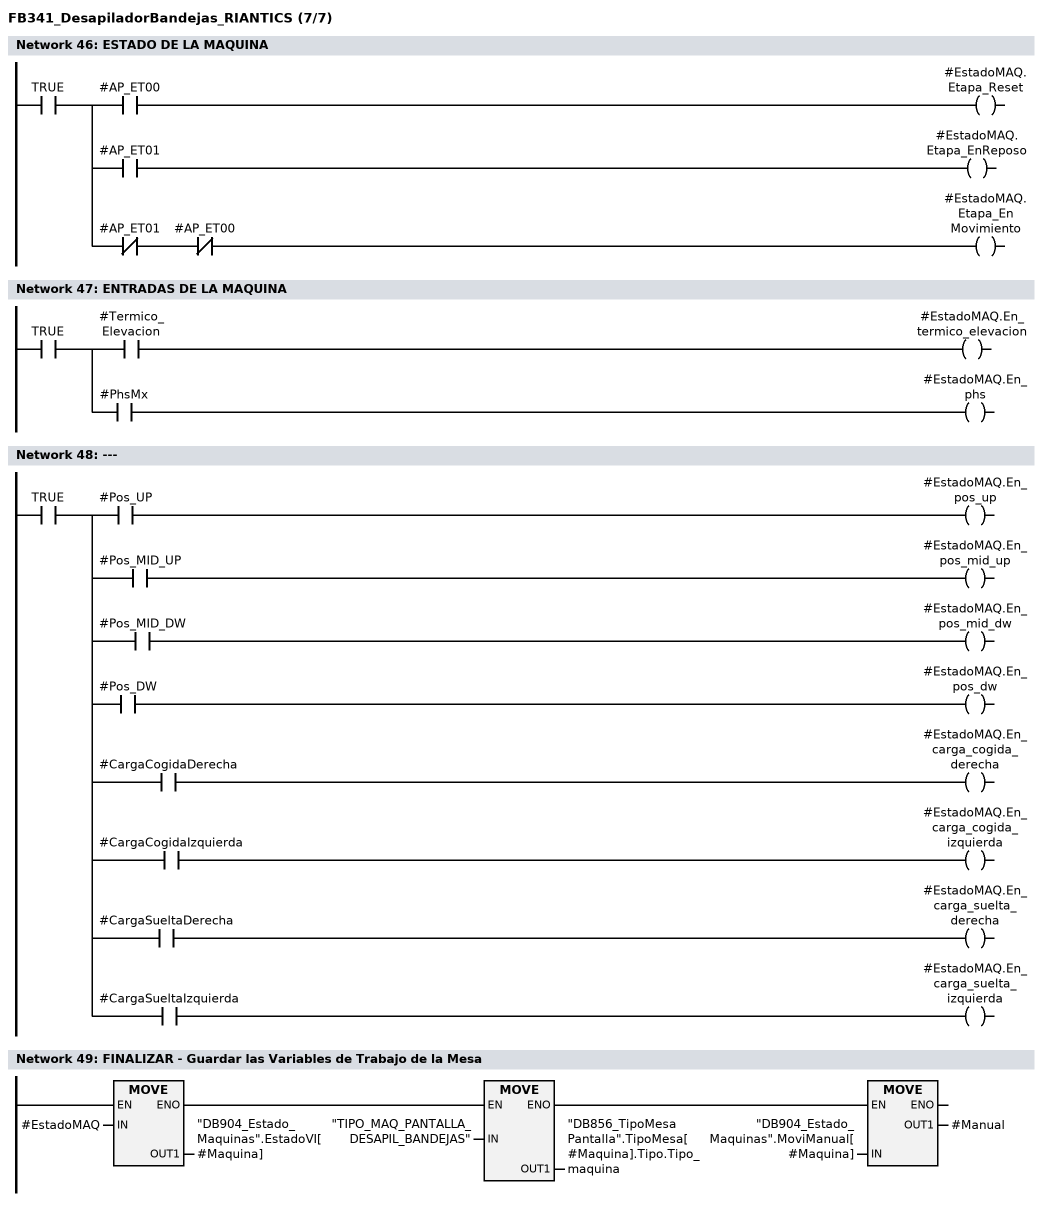
   RUNG wire#powerrail
      Contact( TRUE )
      wire#w1
      Contact( #AP_ET00 )
      Coil( #EstadoMAQ.Etapa_Reset )
   END_RUNG
   RUNG wire#w1
      Contact( #AP_ET01 )
      Coil( #EstadoMAQ.Etapa_EnReposo )
   END_RUNG
   RUNG wire#w1
      I_Contact( #AP_ET01 )
      I_Contact( #AP_ET00 )
      Coil( #EstadoMAQ.Etapa_EnMovimiento )
   END_RUNG
   // the same network as SCL:
   #EstadoMAQ.Etapa_Reset := TRUE AND #AP_ET00;
   #EstadoMAQ.Etapa_EnReposo := TRUE AND #AP_ET01;
   #EstadoMAQ.Etapa_EnMovimiento := TRUE AND NOT #AP_ET01 AND NOT #AP_ET00;
END_REGION

REGION Network 47: ENTRADAS DE LA MAQUINA
   RUNG wire#powerrail
      Contact( TRUE )
      wire#w1
      Contact( #Termico_Elevacion )
      Coil( #EstadoMAQ.En_termico_elevacion )
   END_RUNG
   RUNG wire#w1
      Contact( #PhsMx )
      Coil( #EstadoMAQ.En_phs )
   END_RUNG
   // the same network as SCL:
   #EstadoMAQ.En_termico_elevacion := TRUE AND #Termico_Elevacion;
   #EstadoMAQ.En_phs := TRUE AND #PhsMx;
END_REGION

REGION Network 48: ---
   RUNG wire#powerrail
      Contact( TRUE )
      wire#w1
      Contact( #Pos_UP )
      Coil( #EstadoMAQ.En_pos_up )
   END_RUNG
   RUNG wire#w1
      Contact( #Pos_MID_UP )
      Coil( #EstadoMAQ.En_pos_mid_up )
   END_RUNG
   RUNG wire#w1
      Contact( #Pos_MID_DW )
      Coil( #EstadoMAQ.En_pos_mid_dw )
   END_RUNG
   RUNG wire#w1
      Contact( #Pos_DW )
      Coil( #EstadoMAQ.En_pos_dw )
   END_RUNG
   RUNG wire#w1
      Contact( #CargaCogidaDerecha )
      Coil( #EstadoMAQ.En_carga_cogida_derecha )
   END_RUNG
   RUNG wire#w1
      Contact( #CargaCogidaIzquierda )
      Coil( #EstadoMAQ.En_carga_cogida_izquierda )
   END_RUNG
   RUNG wire#w1
      Contact( #CargaSueltaDerecha )
      Coil( #EstadoMAQ.En_carga_suelta_derecha )
   END_RUNG
   RUNG wire#w1
      Contact( #CargaSueltaIzquierda )
      Coil( #EstadoMAQ.En_carga_suelta_izquierda )
   END_RUNG
   // the same network as SCL:
   #EstadoMAQ.En_pos_up := TRUE AND #Pos_UP;
   #EstadoMAQ.En_pos_mid_up := TRUE AND #Pos_MID_UP;
   #EstadoMAQ.En_pos_mid_dw := TRUE AND #Pos_MID_DW;
   #EstadoMAQ.En_pos_dw := TRUE AND #Pos_DW;
   #EstadoMAQ.En_carga_cogida_derecha := TRUE AND #CargaCogidaDerecha;
   #EstadoMAQ.En_carga_cogida_izquierda := TRUE AND #CargaCogidaIzquierda;
   #EstadoMAQ.En_carga_suelta_derecha := TRUE AND #CargaSueltaDerecha;
   #EstadoMAQ.En_carga_suelta_izquierda := TRUE AND #CargaSueltaIzquierda;
END_REGION

REGION Network 49: FINALIZAR - Guardar las Variables de Trabajo de la Mesa
   RUNG wire#powerrail
      Move(in := #EstadoMAQ, out1 => "DB904_Estado_Maquinas".EstadoVI[#Maquina])
      Move(in := "TIPO_MAQ_PANTALLA_DESAPIL_BANDEJAS", out1 => "DB856_TipoMesaPantalla".TipoMesa[#Maquina].Tipo.Tipo_maquina)
      Move(in := "DB904_Estado_Maquinas".MoviManual[#Maquina], out1 => #Manual)
   END_RUNG
   // the same network as SCL:
   "DB904_Estado_Maquinas".EstadoVI[#Maquina] := #EstadoMAQ;
   "DB856_TipoMesaPantalla".TipoMesa[#Maquina].Tipo.Tipo_maquina := "TIPO_MAQ_PANTALLA_DESAPIL_BANDEJAS";
   #Manual := "DB904_Estado_Maquinas".MoviManual[#Maquina];
END_REGION
END_FUNCTION_BLOCK
